FUNCTION_BLOCK FB2800

 TITLE = 'YieldCalculation'
 //
 // ��Ҫ���ڼ���ࡢ�ꡢ�¡��ղ�����
 // ������ࡢ�аࡢ����ÿ��Сʱ�Ĳ�������
 //
 VERSION: '1.3'
 AUTHOR: QIAO
 NAME:ProCount
 FAMILY:QFam



 //����
 VAR_INPUT
 //ʵʱʵʱƤ�������ۼ���
 Product_Total:REAL;
 //��ʼ���źţ���������Ч��
 Initialize:BOOL;
 END_VAR


  //���
 VAR_OUTPUT

Product_Early_Class:REAL:=0.0;      //��������9:00-17:00��
Product_Middle_Class:REAL:=0.0;    //�а������17:00-1:00��
Product_Late_Class:REAL:=0.0;     //���������1:00-9:00��
Product_Day:REAL:=0.0;           //�ղ���
Product_Month:REAL:=0.0;        //�²���
Product_Year:REAL:=0.0;        //�����
Product_LastMonth:REAL:=0.0;  //���²���
Product_Yesterday:REAL:=0.0; //�������
//���ÿ��Сʱ����
 Product_Early_2H_1:REAL:=0.0;      //����һ��(9:00-11:00)
 Product_Early_2H_2:REAL:=0.0;      //���ڶ���(11:00-13:00)
 Product_Early_2H_3:REAL:=0.0;      //��������(13:00-15:00)
 Product_Early_2H_4:REAL:=0.0;      //�����Ķ�(15:00-17:00)
 //�а�ÿ��Сʱ����
 Product_Middle_2H_1:REAL:=0.0;     //�а��һ��(17:00-19:00)
 Product_Middle_2H_2:REAL:=0.0;     //�а�ڶ���(19:00-21:00)
 Product_Middle_2H_3:REAL:=0.0;     //�а������(21:00-23:00)
 Product_Middle_2H_4:REAL:=0.0;     //�а���Ķ�(23:00-1:00)
 //����ÿ��Сʱ����
 Product_Late_2H_1:REAL:=0.0;      //�����һ��(1:00-3:00)
 Product_Late_2H_2:REAL:=0.0;      //�����ڶ���(3:00-5:00)
 Product_Late_2H_3:REAL:=0.0;      //���������(5:00-7:00)
 Product_Late_2H_4:REAL:=0.0;      //������Ķ�(7:00-9:00)
 //��ʼ����ɱ�־
 Init_Done:BOOL:=FALSE;
 END_VAR

 // Temporary Variables
 VAR_TEMP
           Read_Return :INT ;
 END_VAR

 // Static Variables
 VAR
       //��ǰʱ��
      DateAndTimeNow:DATE_AND_TIME;
      //ʱ��ṹ��
      DateAndTimeNowCoporate AT DateAndTimeNow:STRUCT
      Year:BYTE;
      Month:BYTE;
      Day:BYTE;
      Hour:BYTE;
      Minute:BYTE;
      Second:BYTE;
      milliSecond:WORD;
 END_STRUCT;
     //�洢��ǰʱ�����
      YearNow:INT;
      MonthNow:INT;
      DayNow:INT;
      HourNow:INT;
      MinuteNow:INT;
      SecondNow:INT;
      //�洢��һ��ɨ���ʱ�����
      HourLast:INT;
      MinuteLast:INT;
      SecondLast:INT;
      DayLast:INT;
      MonthLast:INT;
      YearLast:INT;
      //�¡���ʱ��һ�δ洢����
      MonthNowFormer:INT;
      YearNowFormer:INT;
      DayNowFormer:INT;

      //���ࡢ�ա��¡���ʱ��Ĳ���
      StartEarlyClassPro:REAL:=0.0;
      StartMiddleClassPro:REAL:=0.0;
      StartLateClassPro:REAL:=0.0;
      StartDayClassPro:REAL:=0.0;
      StartMonthClassPro:REAL:=0.0;
      StartYearClassPro:REAL:=0.0;
      //���ÿ��Сʱ������ʼֵ
      StartEarly_2H_1:REAL:=0.0; //����һ��(9:00-11:00)
      StartEarly_2H_2:REAL:=0.0; //���ڶ���(11:00-13:00)
      StartEarly_2H_3:REAL:=0.0; //��������(13:00-15:00)
      StartEarly_2H_4:REAL:=0.0; //�����Ķ�(15:00-17:00)
      //�а�ÿ��Сʱ������ʼֵ
      StartMiddle_2H_1:REAL:=0.0; //�а��һ��(17:00-19:00)
      StartMiddle_2H_2:REAL:=0.0; //�а�ڶ���(19:00-21:00)
      StartMiddle_2H_3:REAL:=0.0; //�а������(21:00-23:00)
      StartMiddle_2H_4:REAL:=0.0; //�а���Ķ�(23:00-1:00)
      //����ÿ��Сʱ������ʼֵ
      StartLate_2H_1:REAL:=0.0; //�����һ��(1:00-3:00)
      StartLate_2H_2:REAL:=0.0; //����ڶ���(3:00-5:00)
      StartLate_2H_3:REAL:=0.0; //���������(5:00-7:00)
      StartLate_2H_4:REAL:=0.0; //������Ķ�(7:00-9:00)
      //���ÿ��Сʱ������־λ
      Early_2H_1_Flag:BOOL:=FALSE;
      Early_2H_2_Flag:BOOL:=FALSE;
      Early_2H_3_Flag:BOOL:=FALSE;
      Early_2H_4_Flag:BOOL:=FALSE;
      //�а�ÿ��Сʱ������־λ
      Middle_2H_1_Flag:BOOL:=FALSE;
      Middle_2H_2_Flag:BOOL:=FALSE;
      Middle_2H_3_Flag:BOOL:=FALSE;
      Middle_2H_4_Flag:BOOL:=FALSE;
      //����ÿ��Сʱ������־λ
      Late_2H_1_Flag:BOOL:=FALSE;
      Late_2H_2_Flag:BOOL:=FALSE;
      Late_2H_3_Flag:BOOL:=FALSE;
      Late_2H_4_Flag:BOOL:=FALSE;

      //�״�ɨ���־
      IsFirstScan:BOOL:=TRUE;
      //����־
      EarlyClassFlag:BOOL:=FALSE;
      MiddleClassFlag:BOOL:=FALSE;
      LateClassFlag:BOOL:=FALSE;
      //���������־
      DayFlag:BOOL:=FALSE;
      MonthFlag:BOOL:=FALSE;
      YearFlag:BOOL:=FALSE;
      //���²�����¼
      LastMonth_Total:REAL:=0.0;
      //���������¼
      Yesterday_Total:REAL:=0.0;

 END_VAR

 //�����߼������￪ʼ
 //��ȡϵͳʱ��
 Read_Return:=READ_CLK(CDT :=DateAndTimeNow );
 YearNow:=BCD_TO_INT(DateAndTimeNowCoporate.Year);
 MonthNow:=BCD_TO_INT(DateAndTimeNowCoporate.Month);
 DayNow:=BCD_TO_INT(DateAndTimeNowCoporate.Day);
 HourNow:=BCD_TO_INT(DateAndTimeNowCoporate.Hour);
 MinuteNow:=BCD_TO_INT(DateAndTimeNowCoporate.Minute);
 SecondNow:=BCD_TO_INT(DateAndTimeNowCoporate.Second);

 // �״�ɨ���ʼ��
 IF IsFirstScan THEN
     // ��ʼ�����п�ʼ����Ϊ��ǰ���ۼ���
     StartEarlyClassPro:=Product_Total;
     StartMiddleClassPro:=Product_Total;
     StartLateClassPro:=Product_Total;
     StartDayClassPro:=Product_Total;
     StartMonthClassPro:=Product_Total;
     StartYearClassPro:=Product_Total;
     // ��ʼ�����ÿ��Сʱ������ʼֵ
     StartEarly_2H_1:=Product_Total;
     StartEarly_2H_2:=Product_Total;
     StartEarly_2H_3:=Product_Total;
     StartEarly_2H_4:=Product_Total;
     // ��ʼ���а�ÿ��Сʱ������ʼֵ
     StartMiddle_2H_1:=Product_Total;
     StartMiddle_2H_2:=Product_Total;
     StartMiddle_2H_3:=Product_Total;
     StartMiddle_2H_4:=Product_Total;
     // ��ʼ������ÿ��Сʱ������ʼֵ
     StartLate_2H_1:=Product_Total;
     StartLate_2H_2:=Product_Total;
     StartLate_2H_3:=Product_Total;
     StartLate_2H_4:=Product_Total;
     // ���浱ǰʱ����Ϊ��һ��ɨ��ʱ��
     YearLast:=YearNow;
     MonthLast:=MonthNow;
     DayLast:=DayNow;
     HourLast:=HourNow;
     MinuteLast:=MinuteNow;
     SecondLast:=SecondNow;
     // ���±�־λ
     IsFirstScan:=FALSE;
     Init_Done:=TRUE;
 END_IF;

 // ��ʼ���źŴ���
 IF Initialize THEN
     // �������п�ʼ����Ϊ��ǰ���ۼ���
     StartEarlyClassPro:=Product_Total;
     StartMiddleClassPro:=Product_Total;
     StartLateClassPro:=Product_Total;
     StartDayClassPro:=Product_Total;
     StartMonthClassPro:=Product_Total;
     StartYearClassPro:=Product_Total;
     // �������ÿ��Сʱ������ʼֵ
     StartEarly_2H_1:=Product_Total;
     StartEarly_2H_2:=Product_Total;
     StartEarly_2H_3:=Product_Total;
     StartEarly_2H_4:=Product_Total;
     // �����а�ÿ��Сʱ������ʼֵ
     StartMiddle_2H_1:=Product_Total;
     StartMiddle_2H_2:=Product_Total;
     StartMiddle_2H_3:=Product_Total;
     StartMiddle_2H_4:=Product_Total;
     // ��������ÿ��Сʱ������ʼֵ
     StartLate_2H_1:=Product_Total;
     StartLate_2H_2:=Product_Total;
     StartLate_2H_3:=Product_Total;
     StartLate_2H_4:=Product_Total;
     // �������в���Ϊ0
     Product_Early_Class:=0.0;
     Product_Middle_Class:=0.0;
     Product_Late_Class:=0.0;
     Product_Day:=0.0;
     Product_Month:=0.0;
     Product_Year:=0.0;
     // �������ÿ��Сʱ����Ϊ0
     Product_Early_2H_1:=0.0;
     Product_Early_2H_2:=0.0;
     Product_Early_2H_3:=0.0;
     Product_Early_2H_4:=0.0;
     // �����а�ÿ��Сʱ����Ϊ0
     Product_Middle_2H_1:=0.0;
     Product_Middle_2H_2:=0.0;
     Product_Middle_2H_3:=0.0;
     Product_Middle_2H_4:=0.0;
     // ��������ÿ��Сʱ����Ϊ0
     Product_Late_2H_1:=0.0;
     Product_Late_2H_2:=0.0;
     Product_Late_2H_3:=0.0;
     Product_Late_2H_4:=0.0;
     // ���±�־λ
     Init_Done:=TRUE;
 END_IF;

 // ���������㣨9:00-17:00��
 // �ж��Ƿ�������ʱ�䣨9:00:00��
 IF (HourNow =9 AND MinuteNow=0 AND SecondNow=0) OR
    (HourLast <9 AND HourNow>=9) THEN // ������Сʱ�����
     StartEarlyClassPro:=Product_Total;
     EarlyClassFlag:=TRUE;
 END_IF;

 // �ж��Ƿ��˳����ʱ�䣨17:00:00��
 IF (HourNow =17 AND MinuteNow=0 AND SecondNow=0) OR
    (HourLast <17 AND HourNow>=17) THEN // ������Сʱ�����
     EarlyClassFlag:=FALSE;
 END_IF;

 // ����������
 IF HourNow>=9 AND HourNow<17 THEN
    Product_Early_Class:=Product_Total - StartEarlyClassPro;
 END_IF;

 // ���ÿ��Сʱ��������
 // ����һ��(9:00-11:00)
 IF (HourNow =9 AND MinuteNow=0 AND SecondNow=0) OR
    (HourLast <9 AND HourNow>=9) THEN
     StartEarly_2H_1:=Product_Total;
     Early_2H_1_Flag:=TRUE;
 END_IF;

 IF (HourNow =11 AND MinuteNow=0 AND SecondNow=0) OR
    (HourLast <11 AND HourNow>=11) THEN
     Early_2H_1_Flag:=FALSE;
 END_IF;

 IF HourNow>=9 AND HourNow<11 THEN
    Product_Early_2H_1:=Product_Total - StartEarly_2H_1;
 END_IF;

 // ���ڶ���(11:00-13:00)
 IF (HourNow =11 AND MinuteNow=0 AND SecondNow=0) OR
    (HourLast <11 AND HourNow>=11) THEN
     StartEarly_2H_2:=Product_Total;
     Early_2H_2_Flag:=TRUE;
 END_IF;

 IF (HourNow =13 AND MinuteNow=0 AND SecondNow=0) OR
    (HourLast <13 AND HourNow>=13) THEN
     Early_2H_2_Flag:=FALSE;
 END_IF;

 IF HourNow>=11 AND HourNow<13 THEN
    Product_Early_2H_2:=Product_Total - StartEarly_2H_2;
 END_IF;

 // ��������(13:00-15:00)
 IF (HourNow =13 AND MinuteNow=0 AND SecondNow=0) OR
    (HourLast <13 AND HourNow>=13) THEN
     StartEarly_2H_3:=Product_Total;
     Early_2H_3_Flag:=TRUE;
 END_IF;

 IF (HourNow =15 AND MinuteNow=0 AND SecondNow=0) OR
    (HourLast <15 AND HourNow>=15) THEN
     Early_2H_3_Flag:=FALSE;
 END_IF;

 IF HourNow>=13 AND HourNow<15 THEN
    Product_Early_2H_3:=Product_Total - StartEarly_2H_3;
 END_IF;

 // �����Ķ�(15:00-17:00)
 IF (HourNow =15 AND MinuteNow=0 AND SecondNow=0) OR
    (HourLast <15 AND HourNow>=15) THEN
     StartEarly_2H_4:=Product_Total;
     Early_2H_4_Flag:=TRUE;
 END_IF;

 IF (HourNow =17 AND MinuteNow=0 AND SecondNow=0) OR
    (HourLast <17 AND HourNow>=17) THEN
     Early_2H_4_Flag:=FALSE;
 END_IF;

 IF HourNow>=15 AND HourNow<17 THEN
    Product_Early_2H_4:=Product_Total - StartEarly_2H_4;
 END_IF;

 // �а�������㣨17:00-1:00��
 // �ж��Ƿ�����а�ʱ�䣨17:00:00��
 IF (HourNow =17 AND MinuteNow=0 AND SecondNow=0) OR
    (HourLast <17 AND HourNow>=17) THEN // ������Сʱ�����
     StartMiddleClassPro:=Product_Total;
     MiddleClassFlag:=TRUE;
 END_IF;

 // �ж��Ƿ��˳��а�ʱ�䣨1:00:00��
 IF (HourNow =1 AND MinuteNow=0 AND SecondNow=0) OR
    (HourLast >=17) THEN // ������������
     MiddleClassFlag:=FALSE;
 END_IF;

 // �����а����
 IF (HourNow>=17 AND HourNow<=23) OR (HourNow>=0 AND HourNow<1) THEN
     Product_Middle_Class:=Product_Total - StartMiddleClassPro;
 END_IF;

 // �а�ÿ��Сʱ��������
 // �а��һ��(17:00-19:00)
 IF (HourNow =17 AND MinuteNow=0 AND SecondNow=0) OR
    (HourLast <17 AND HourNow>=17) THEN
     StartMiddle_2H_1:=Product_Total;
     Middle_2H_1_Flag:=TRUE;
 END_IF;

 IF (HourNow =19 AND MinuteNow=0 AND SecondNow=0) OR
    (HourLast <19 AND HourNow>=19) THEN
     Middle_2H_1_Flag:=FALSE;
 END_IF;

 IF HourNow>=17 AND HourNow<19 THEN
    Product_Middle_2H_1:=Product_Total - StartMiddle_2H_1;
 END_IF;

 // �а�ڶ���(19:00-21:00)
 IF (HourNow =19 AND MinuteNow=0 AND SecondNow=0) OR
    (HourLast <19 AND HourNow>=19) THEN
     StartMiddle_2H_2:=Product_Total;
     Middle_2H_2_Flag:=TRUE;
 END_IF;

 IF (HourNow =21 AND MinuteNow=0 AND SecondNow=0) OR
    (HourLast <21 AND HourNow>=21) THEN
     Middle_2H_2_Flag:=FALSE;
 END_IF;

 IF HourNow>=19 AND HourNow<21 THEN
    Product_Middle_2H_2:=Product_Total - StartMiddle_2H_2;
 END_IF;

 // �а������(21:00-23:00)
 IF (HourNow =21 AND MinuteNow=0 AND SecondNow=0) OR
    (HourLast <21 AND HourNow>=21) THEN
     StartMiddle_2H_3:=Product_Total;
     Middle_2H_3_Flag:=TRUE;
 END_IF;

 IF (HourNow =23 AND MinuteNow=0 AND SecondNow=0) OR
    (HourLast <23 AND HourNow>=23) THEN
     Middle_2H_3_Flag:=FALSE;
 END_IF;

 IF HourNow>=21 AND HourNow<23 THEN
    Product_Middle_2H_3:=Product_Total - StartMiddle_2H_3;
 END_IF;

 // �а���Ķ�(23:00-1:00)
 IF (HourNow =23 AND MinuteNow=0 AND SecondNow=0) OR
    (HourLast <23 AND HourNow>=23) THEN
     StartMiddle_2H_4:=Product_Total;
     Middle_2H_4_Flag:=TRUE;
 END_IF;

 IF (HourNow =1 AND MinuteNow=0 AND SecondNow=0) OR
    (HourLast >=23) THEN
     Middle_2H_4_Flag:=FALSE;
 END_IF;

 IF (HourNow>=23 AND HourNow<=23) OR (HourNow>=0 AND HourNow<1) THEN
    Product_Middle_2H_4:=Product_Total - StartMiddle_2H_4;
 END_IF;

 // ����������㣨1:00-9:00��
 // �ж��Ƿ��������ʱ�䣨1:00:00��
 IF (HourNow =1 AND MinuteNow=0 AND SecondNow=0) OR
    (HourLast >=17) THEN // ������������
     StartLateClassPro:=Product_Total;
     LateClassFlag:=TRUE;
 END_IF;

 // �ж��Ƿ��˳�����ʱ�䣨9:00:00��
 IF (HourNow =9 AND MinuteNow=0 AND SecondNow=0) OR
    (HourLast <9 AND HourNow>=9) THEN // ������Сʱ�����
     LateClassFlag:=FALSE;
 END_IF;

 // �����������
 IF HourNow>=1 AND HourNow<9 THEN
     Product_Late_Class:=Product_Total - StartLateClassPro;
 END_IF;

 // ����ÿ��Сʱ��������
 // �����һ��(1:00-3:00)
 IF (HourNow =1 AND MinuteNow=0 AND SecondNow=0) OR
    (HourLast >=17) THEN
     StartLate_2H_1:=Product_Total;
     Late_2H_1_Flag:=TRUE;
 END_IF;

 IF (HourNow =3 AND MinuteNow=0 AND SecondNow=0) OR
    (HourLast <3 AND HourNow>=3) THEN
     Late_2H_1_Flag:=FALSE;
 END_IF;

 IF HourNow>=1 AND HourNow<3 THEN
    Product_Late_2H_1:=Product_Total - StartLate_2H_1;
 END_IF;

 // ����ڶ���(3:00-5:00)
 IF (HourNow =3 AND MinuteNow=0 AND SecondNow=0) OR
    (HourLast <3 AND HourNow>=3) THEN
     StartLate_2H_2:=Product_Total;
     Late_2H_2_Flag:=TRUE;
 END_IF;

 IF (HourNow =5 AND MinuteNow=0 AND SecondNow=0) OR
    (HourLast <5 AND HourNow>=5) THEN
     Late_2H_2_Flag:=FALSE;
 END_IF;

 IF HourNow>=3 AND HourNow<5 THEN
    Product_Late_2H_2:=Product_Total - StartLate_2H_2;
 END_IF;

 // ���������(5:00-7:00)
 IF (HourNow =5 AND MinuteNow=0 AND SecondNow=0) OR
    (HourLast <5 AND HourNow>=5) THEN
     StartLate_2H_3:=Product_Total;
     Late_2H_3_Flag:=TRUE;
 END_IF;

 IF (HourNow =7 AND MinuteNow=0 AND SecondNow=0) OR
    (HourLast <7 AND HourNow>=7) THEN
     Late_2H_3_Flag:=FALSE;
 END_IF;

 IF HourNow>=5 AND HourNow<7 THEN
    Product_Late_2H_3:=Product_Total - StartLate_2H_3;
 END_IF;

 // ������Ķ�(7:00-9:00)
 IF (HourNow =7 AND MinuteNow=0 AND SecondNow=0) OR
    (HourLast <7 AND HourNow>=7) THEN
     StartLate_2H_4:=Product_Total;
     Late_2H_4_Flag:=TRUE;
 END_IF;

 IF (HourNow =9 AND MinuteNow=0 AND SecondNow=0) OR
    (HourLast <9 AND HourNow>=9) THEN
     Late_2H_4_Flag:=FALSE;
 END_IF;

 IF HourNow>=7 AND HourNow<9 THEN
    Product_Late_2H_4:=Product_Total - StartLate_2H_4;
 END_IF;

 // �ղ������㣨9:00-����9:00��
 // �ж��Ƿ�����µ�һ�죨9:00:00��
 IF (HourNow =9 AND MinuteNow=0 AND SecondNow=0) OR
    (HourLast <9 AND HourNow>=9) THEN // ������Сʱ�����
     StartDayClassPro:=Product_Total;
     DayFlag:=TRUE;
 END_IF;

 // �����ղ���
Product_Day:=Product_Total - StartDayClassPro;

// ��¼������������µ�һ�쿪ʼʱ��
IF DayFlag THEN
    // ��������Ĳ���
    Yesterday_Total := Product_Day;
    // �������Ĳ���
    Product_Yesterday := Yesterday_Total;
    // �����ձ�־
    DayFlag := FALSE;
END_IF;

 // �²������㣨ÿ��1��9:00��ʼ��
 // �ж��Ƿ�����µ�һ�£�1��9:00:00��
 IF (DayNow=1 AND HourNow>=9) AND
    (DayLast>1 OR (DayLast=1 AND HourLast<9)) THEN // �������ջ��Сʱ�����
     StartMonthClassPro:=Product_Total;
     MonthFlag:=TRUE;
 END_IF;

 // �����²���
Product_Month:=Product_Total - StartMonthClassPro;

// ��¼���²��������µ�һ�¿�ʼʱ��
IF MonthFlag THEN
    // �������µĲ���
    LastMonth_Total := Product_Month;
    // ������µĲ���
    Product_LastMonth := LastMonth_Total;
    // �����±�־
    MonthFlag := FALSE;
END_IF;

 // ��������㣨ÿ��1��1��9:00��ʼ��
 // �ж��Ƿ�����µ�һ�꣨1��1��9:00:00��
 IF (MonthNow=1 AND DayNow=1 AND HourNow>=9) AND
    ((MonthLast>1) OR (MonthLast=1 AND DayLast>1) OR (MonthLast=1 AND DayLast=1 AND HourLast<9)) THEN // �������ꡢ���»��Сʱ�����
     StartYearClassPro:=Product_Total;
     YearFlag:=TRUE;
 END_IF;

 // ���������
 Product_Year:=Product_Total - StartYearClassPro;

 // ���浱ǰʱ����Ϊ��һ��ɨ�����һ��ʱ��
 YearLast:=YearNow;
 MonthLast:=MonthNow;
 DayLast:=DayNow;
 HourLast:=HourNow;
 MinuteLast:=MinuteNow;
 SecondLast:=SecondNow;

 END_FUNCTION_BLOCK

DATA_BLOCK DB2800 FB2800
 BEGIN
 END_DATA_BLOCK